(* PLC project flask_motion_app_copy, Dassault Systèmes ControlBuild 2024x Refresh1 *)
(* stored: creationDateTime 2024-04-15T17:56:08-01:00 *)

PROGRAM flask_motion_app.flask_motion_app_copy
  VAR_INPUT
    weight : INT := 150;
  END_VAR
  VAR_OUTPUT
    masterPosition : REAL := 0.0;
  END_VAR

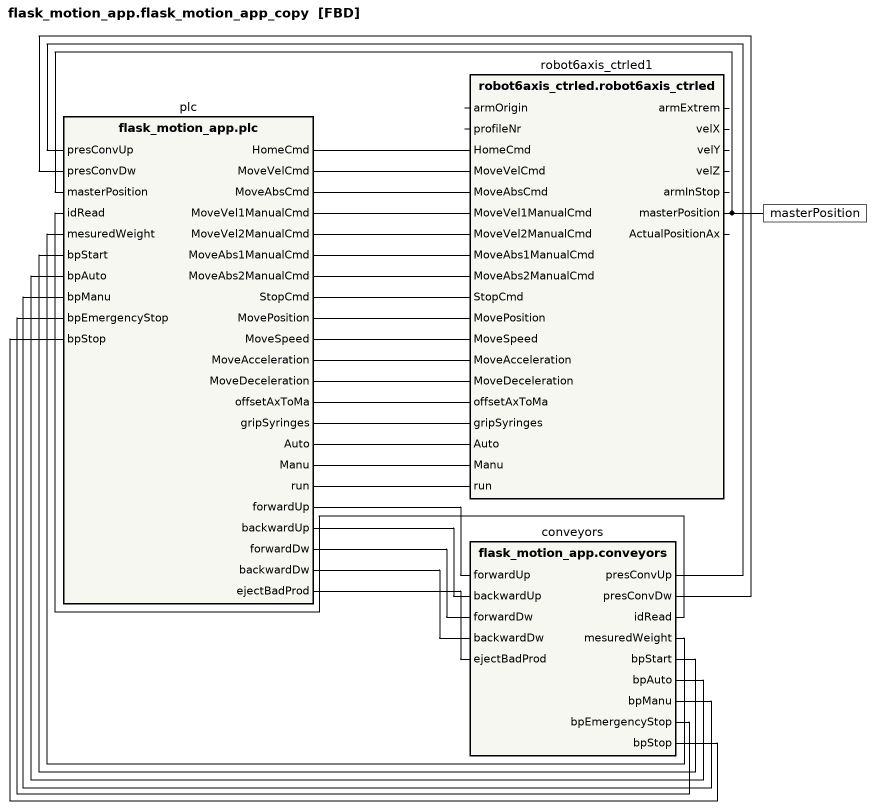
(* FBD diagram, written out as Structured Text *)
conveyors(forwardUp := plc.forwardUp, backwardUp := plc.backwardUp, forwardDw := plc.forwardDw, backwardDw := plc.backwardDw, ejectBadProd := plc.ejectBadProd);
plc(presConvUp := conveyors.presConvUp, presConvDw := conveyors.presConvDw, masterPosition := robot6axis_ctrled1.masterPosition, idRead := conveyors.idRead, mesuredWeight := conveyors.mesuredWeight, bpStart := conveyors.bpStart, bpAuto := conveyors.bpAuto, bpManu := conveyors.bpManu, bpEmergencyStop := conveyors.bpEmergencyStop, bpStop := conveyors.bpStop);
robot6axis_ctrled1(HomeCmd := plc.HomeCmd, MoveVelCmd := plc.MoveVelCmd, MoveAbsCmd := plc.MoveAbsCmd, MoveVel1ManualCmd := plc.MoveVel1ManualCmd, MoveVel2ManualCmd := plc.MoveVel2ManualCmd, MoveAbs1ManualCmd := plc.MoveAbs1ManualCmd, MoveAbs2ManualCmd := plc.MoveAbs2ManualCmd, StopCmd := plc.StopCmd, MovePosition := plc.MovePosition, MoveSpeed := plc.MoveSpeed, MoveAcceleration := plc.MoveAcceleration, MoveDeceleration := plc.MoveDeceleration, offsetAxToMa := plc.offsetAxToMa, gripSyringes := plc.gripSyringes, Auto := plc.Auto, Manu := plc.Manu, run := plc.run);
masterPosition := robot6axis_ctrled1.masterPosition;
END_PROGRAM
